// TIA Portal V21 export
TYPE "motorConfig"
   STRUCT
      almMask : Word := 16#07FF;
      fbDelayMax { S7_SetPoint := 'True'} : Time := T#3s;
      restartDelay : Time := T#10s;
      minSpeedSp : Real := 0.0;
      maxSpeedSp : Real := 1000.0;
      minOnTime : Time := T#2s;
   END_STRUCT;
END_TYPE
